# EPICS substitutions: iocBoot/ioc14idc/iocEnvVar.substitutions
#==============================================================================
#
# Abs:  IOC Administration Records
#
# Name: iocAdmin.substitutions
#
#==============================================================================
# Edited to work at BioCARS.

file "$(DEVIOCSTATS)/db/iocEnvVar.db"
{
pattern { IOCNAME, ENVNAME      , ENVVAR                          , ENVTYPE}
	{ 14IDC , LOCATION     , LOCATION                        , env    }
	{ 14IDC , ENGINEER     , ENGINEER                        , env    }
	{ 14IDC , CA_ADDR_LIST , EPICS_CA_ADDR_LIST              , epics  }
	{ 14IDC , CA_CONN_TIME , EPICS_CA_CONN_TMO               , epics  }
	{ 14IDC , CA_AUTO_ADDR , EPICS_CA_AUTO_ADDR_LIST         , epics  }
	{ 14IDC , CA_RPTR_PORT , EPICS_CA_REPEATER_PORT          , epics  }
	{ 14IDC , CA_SRVR_PORT , EPICS_CA_SERVER_PORT            , epics  }
	{ 14IDC , CA_MAX_ARRAY , EPICS_CA_MAX_ARRAY_BYTES        , epics  }
	{ 14IDC , CA_SRCH_TIME , EPICS_CA_MAX_SEARCH_PERIOD      , epics  }
	{ 14IDC , CA_BEAC_TIME , EPICS_CA_BEACON_PERIOD          , epics  }
	{ 14IDC , TIMEZONE     , EPICS_TIMEZONE                  , epics  }
	{ 14IDC , TS_NTP_INET  , EPICS_TS_NTP_INET               , epics  }
	{ 14IDC , IOC_LOG_PORT , EPICS_IOC_LOG_PORT              , epics  }
	{ 14IDC , IOC_LOG_INET , EPICS_IOC_LOG_INET              , epics  }
}
